Omron CX-Programmer project NewProject (CX-Programmer 9.70)

# PLC NewPLC1: CP1E E20

## Global symbols (name address type ; comment)
0.00 BOOL  ; start
0.01 BOOL  ; nc
0.02 BOOL  ; start
100.00 BOOL  ; led

## Program NewProgram1 (cyclic task 0)

### Section Section1

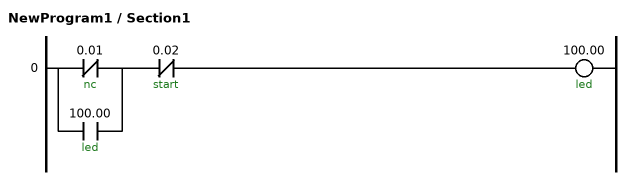
; rung 0
LDNOT 0.01  ; nc
OR 100.00  ; led
ANDNOT 0.02  ; start
OUT 100.00  ; led

### Section END
; rung 0
END(001)